Fanuc KAREL source: kt00268.KL

-- PROVISIONAL review KL for V1013-1; original PC SHA256 3fec7dcf6c8f1cfaddeaf0b390d068c76507e61fb2fad8a3d53532275baf5bbb
-- Incomplete behavior may be omitted. Consult companion uncertainty JSON. Do not deploy.
PROGRAM KT00268
%NOLOCKGROUP
VAR
  R2 : REAL
  OUT : BOOLEAN
-- UNRESOLVED_DECL Y1 type=002018
BEGIN
  -- UNRESOLVED_PC offsets 5-19; opcodes 2E,22,9D,33,B2
  -- UNRESOLVED_PC offsets 24-35; opcodes 2E,23
  -- UNRESOLVED_PC offsets 40-64; opcodes 22,9D,33,B1,21,29,64,6D,23
  -- UNRESOLVED_PC offsets 69-73; opcodes 7F
END KT00268
